(* CoDeSys 2.3.9.35 project: Exercício 8.pro *)
(* Author: Altus *)
(* Libraries: DU35x.lib 7.7.11 15:59:13, Navigation.lib 15.7.11 10:06:00, SysLibTargetVisu.lib 26.11.08 09:53:28, Standard.lib 26.11.08 09:46:20, Iecsfc.lib 26.11.08 09:46:14, SYSLIBCALLBACK.LIB 26.11.08 09:53:30 *)

(* PLC configuration (modules and I/O channels)
Configuração do CP [Root] node -1, in %IB0 out %QB0
  Comunicação [Comunica] node 0, in %IB0 out %QB0
    COM1 [COM1] node 0, in %IB0 out %QB0 {BaudRate = 115200; Paridade = Sem Paridade; StopBits = 1 Stop Bit; Modem = Sem RTS/CTS; Delay = 5}
      MToolIEC [Codesys] node 0, in %IB0 out %QB0
    COM2 [COM2] node 1, in %IB0 out %QB0 {BaudRate = 115200; Paridade = Sem Paridade; StopBits = 1 Stop Bit; Modem = Sem RTS/CTS; Delay = 5}
      Desabilitada [Desabilitado485] node 0, in %IB0 out %QB0
  Barramento [Barramento] node 1, in %IB0 out %QB0
    Entradas [Entradas] node 0, in %IB0 out %QB0
      Entradas Digitais 0 [Entradas0] node 0, in %IW0 out %QB0
        I00 AT %IX0.0 [BitInput] I0.0
        I01 AT %IX0.1 [BitInput] I0.1
        I02 AT %IX0.2 [BitInput] I0.2
        I03 AT %IX0.3 [BitInput] I0.3
        I04 AT %IX0.4 [BitInput] I0.4
        I05 AT %IX0.5 [BitInput] I0.5
        I06 AT %IX0.6 [BitInput] I0.6
        I07 AT %IX0.7 [BitInput] I0.7
        I08 AT %IX0.8 [BitInput] I0.8
      Entradas Digitais 1 [Entradas1] node 0, in %IW1 out %QB0
        I10 AT %IX1.0 [BitInput] I1.0
        I11 AT %IX1.1 [BitInput] I1.1
        I12 AT %IX1.2 [BitInput] I1.2
        I13 AT %IX1.3 [BitInput] I1.3
        I14 AT %IX1.4 [BitInput] I1.4
        I15 AT %IX1.5 [BitInput] I1.5
        I16 AT %IX1.6 [BitInput] I1.6
        I17 AT %IX1.7 [BitInput] I1.7
        I18 AT %IX1.8 [BitInput] I1.8
      Entradas Digitais 2 [Entradas2] node 0, in %IW2 out %QB0
        I20 AT %IX2.0 [BitInput] I2.0
        I21 AT %IX2.1 [BitInput] I2.1
      Entradas Analógicas [EntradaAnalogica] node 0, in %IW4 out %QB0
        AI0 AT %IW4 [WordInput] AI0 {TipoAnalogica = Channel Disable; FiltroAnalogica = Filter 0 - AI=2ms  / AV=90ms; FundoEscala = 0}
        AI1 AT %IW5 [WordInput] AI1 {TipoAnalogica = Channel Disable; FiltroAnalogica = Filter 0 - AI=2ms  / AV=90ms; FundoEscala = 0}
        AI2 AT %IW6 [WordInput] AI2 {TipoAnalogica = Channel Disable; FiltroAnalogica = Filter 0 - AI=2ms  / AV=90ms; FundoEscala = 0}
        AI3 AT %IW7 [WordInput] AI3 {TipoAnalogica = Channel Disable; FiltroAnalogica = Filter 0 - AI=2ms  / AV=90ms; FundoEscala = 0}
      Entradas Rápidas [EntradasRapidas] node 1, in %IB16 out %QB0
        Bloco 0 [Bloco0] node 0, in %IB16 out %QB0
          Desabilitado [DesabilitadoBloco0] node 0, in %IB16 out %QB0
        Bloco 1 [Bloco1] node 1, in %IB16 out %QB0
          Desabilitado [DesabilitadoBloco1] node 0, in %IB16 out %QB0
        Entrada Configuravél Bloco 0 [EntradaConfiBloco0] node 2, in %IB16 out %QB0
          Contador 0 [EntradaConfContador0] node 0, in %IB16 out %QB0 {EntradaConfiguravelContador = Disable}
        Entrada Configuravél Bloco 1 [EntradaConfiBloco1] node 3, in %IB16 out %QB0
          Contador 2 [EntradaConfContador2] node 0, in %IB16 out %QB0 {EntradaConfiguravelContador = Disable}
    Saídas [Saidas] node 1, in %IB13 out %QB0
      Saídas Digitais 0 [Saidas0] node 0, in %IW0 out %QW0
        Q00 AT %QX0.0 [BitOutput] Q0.0
        Q01 AT %QX0.1 [BitOutput] Q0.1
        Q02 AT %QX0.2 [BitOutput] Q0.2
        Q03 AT %QX0.3 [BitOutput] Q0.3
        Q04 AT %QX0.4 [BitOutput] Q0.4
        Q05 AT %QX0.5 [BitOutput] Q0.5
        Q06 AT %QX0.6 [BitOutput] Q0.6
        Q07 AT %QX0.7 [BitOutput] Q0.7
      Saídas Digitais 1 [Saidas1] node 0, in %IW0 out %QW1
        Q10 AT %QX1.0 [BitOutput] Q1.0
        Q11 AT %QX1.1 [BitOutput] Q1.1
        Q12 AT %QX1.2 [BitOutput] Q1.2
        Q13 AT %QX1.3 [BitOutput] Q1.3
        Q14 AT %QX1.4 [BitOutput] Q1.4
        Q15 AT %QX1.5 [BitOutput] Q1.5
        Q16 AT %QX1.6 [BitOutput] Q1.6
        Q17 AT %QX1.7 [BitOutput] Q1.7
      Saídas Analógicas [SaidaAnalogica] node 0, in %IW0 out %QW3
        AO0 AT %QW3 [WordOutput] AO0 {TipoAnalogica = Channel Disable; FundoEscala = 0}
        AO1 AT %QW4 [WordOutput] AO1 {TipoAnalogica = Channel Disable; FundoEscala = 0}
      Saídas Rápidas [SaidasRapidas] node 1, in %IB0 out %QB10
        Saída Rápida 0 Desabilitada [DesabilitadoF0] node 0, in %IB0 out %QB10
        Saída Rápida 1 Desabilitada [DesabilitadoF1] node 1, in %IB0 out %QB10
      Saídas Comum de Contador [SaidasContador] node 2, in %IB0 out %QB10
        Saída do Bloco 0 Desabilitada [DesabilitadoSaidaBloco0] node 0, in %IB0 out %QB10
        Saída do Bloco 1 Desabilitada [DesabilitadoSaidaBloco1] node 1, in %IB0 out %QB10
  Eventos Externos [Eventos] node 2, in %IB13 out %QB6
    Evento Temporizado [TimerEvent] node 0, in %IB13 out %QB6 {Intervalo = 10}
*)

(* Task configuration *)
TASK PRINCIPAL (PRIORITY := 1, INTERVAL := T#1ms);
	PLC_PRG();
END_TASK
TASK NAVIGATION (PRIORITY := 1, INTERVAL := T#20ms);
	NAVEGA();
END_TASK
TASK VISUALIZATION (PRIORITY := 1, INTERVAL := T#500ms);
	MAINTARGETVISU_PAINT_CODE
END_TASK
TASK KEYBOARD_USAGE (PRIORITY := 1, INTERVAL := T#20ms);
	MAINTARGETVISU_INPUT_CODE
END_TASK

(* POU PLC_PRG, ST *)
(*Um fulão processa o couro através do seguinte procedimento: A partir de um botão de início (entrada digital):
a) Inicialmente, preenche-se o fulão com o produto de curtimento, através da válvula VPC.
b) O motor é acionado no sentido horário, através da saída MH por um tempo THC.
c) O motor é acionado no sentido anti-horário, através da saída MAH, por um tempo TAHC.
d) O fulão é esvaziado, através da válvula VD.
e) O fulão é preenchido com água, através da válvula VL.
f) O motor é acionado no sentido horário, através da saída MH por um tempo THL.
g) O motor é acionado no sentido anti-horário, através da saída MAH, por um tempo TAHL.
h) O fulão é esvaziado, através da válvula VD.
i) É sinalizado, através de uma lâmpada FP, o final do processo.
Após o ciclo completo, o sistema deve ficar pronto para ser acionado novamente. O nível alto do fulão é indicado pela chave de
nível NVC, e o nível baixo (vazio) é indicado pela chave NVV. Elabore um programa que realize este procedimento, com os 
seguintes tempos para simulação: THC =TAHC= 5s. THL=TAHL=8s
Cada fase do processo deve ser devidamente apresentada na tela da IHM através de uma variável de texto.*)


PROGRAM PLC_PRG
VAR
	START AT %IX0.0: BOOL;
	NVC AT %IX0.1: BOOL; (*válvula que indica o nível alto do fulão*)
	NVV AT %IX0.2: BOOL; (*válvula que indica o nível baixo do fulão*)
	VPC AT %QX1.0: BOOL; (*válvula que inicia o preenchimento do fulão com produto de curtimento*)
	MH AT %QX1.1: BOOL; (*gira o motor no sentido horário*)
	MAH AT %QX1.2: BOOL; (*gira o motor no sentido anti-horário*)
	VD AT %QX1.3: BOOL; (*válvula que esvazia o fulão*)
	VL AT %QX1.4: BOOL; (*válvula que preenche o fulão com água*)
	FP AT %QX1.5: BOOL := 1; (*lâmpada que sinaliza quando o processo termina, começa acesa*)
	THC: TIME := T#5s; (*tempo que o motor fica girando no sentido horário, quando está esvaziando o fulão*)
	TAHC: TIME := T#5s; (*tempo que o motor fica girando no sentido anti-horário, quando está esvaziando o fulão*)
	THL: TIME := T#8s; (*tempo que o motor fica girando no sentido horário, quando está enchendo o fulão*)
	TAHL: TIME := T#8s; (*tempo que o motor fica girando no sentido anti-horário, quando está enchendo o fulão*)
	TH: TIME;
	TAH: TIME;
	T1: TON;
	T2: TON;
	B0: R_TRIG; (*borda de subida do botão de START*)
	B1: R_TRIG; (*borda de subida de NVC, que significa que chegou no nível alto do fulão*)
	B2: R_TRIG; (*borda de subida de NVV, que significa que chegou no nível baixo do fulão*)
	M1: INT := 0; (*variável de controle para o programa*)
	MSG: STRING(50) := 'DESLIGADO';
END_VAR
T1(IN := MH, PT := TH);
T2(IN := MAH, PT := TAH);
B0(CLK := START); (*borda de subida do botão de START*)
B1(CLK := NVC); (*borda de subida de NVC, que significa que chegou no nível ALTO do fulão*)
B2(CLK := NVV); (*borda de subida de NVV, que significa que chegou no nível BAIXO do fulão*)

IF B0.Q AND FP THEN (*quando der a borda de subida do botão de START*)
	FP := 0; (*desliga a lâmpada de FP, pois o processo se inicializou*)
	M1 := 1; (*iguala M1 a 1, que será usado depois*)
	VPC := 1; (*começa a enxer a válvula VPC, preenchendo o fulão com o produto de curtimento*)
	MSG := 'ENCHENDO O FULÃO COM PRODUTO DE CURTIMENTO';
END_IF

IF NOT FP THEN (*se a lâmpada estiver desligada, ou seja, não terminou o processo*)
	IF B1.Q THEN (*se chegou no nível alto do fulão*)
		IF VL THEN (*preencheu o fulão com água através da válvula VL*)
			VL := 0; (*desliga a válvula de água*)
			TH := THL; (*iguala o tempo de TH ao de THL, que é de 8 segundos*)
			TAH := TAHL; (*iguala o tempo de TAH ao de TAHL, que é de 8 segundos*)
		ELSE (*se encheu de produto de curtimento*)
			VPC := 0; (*desliga a válvula VPC de produto de curtimento, que para de mandar líquido para o fulão*)
			TH := THC; (*iguala o tempo de TH ao de THC, que é de 5 segundos*)
			TAH := TAHC; (*iguala o tempo de TAH ao de TAHC, que é de 5 segundos*)
		END_IF
		MH := 1; (*gira o motor no sentido horário por x segundos*)
		MSG := 'MOTOR GIRANDO NO SENTIDO HORÁRIO';
	END_IF
	IF T1.Q THEN (*quando acabar de contar o tempo de TH e der verdadeiro na saída T1.Q*)
		MH := 0; (*desliga a saída de MH*)
		MAH := 1; (*e aciona o motor no sentido anti-horário com a saída MAH por x segundos*)
		MSG := 'MOTOR GIRANDO NO SENTIDO ANTI-HORÁRIO';
	END_IF
	IF T2.Q THEN (*quando acabar de contar o tempo de TAHL e der verdadeiro na saída T2.Q*)
		MAH := 0; (*desliga a saída de MAH*)
		VD := 1; (*esvazia o fulão através da válvula VD*)
		MSG := 'ESVAZIANDO O FULÃO';
	END_IF
	IF B2.Q THEN (*se chegou no nível baixo do fulão*)
		VD := 0; (*desliga a válvula VD, para parar de esvaziar o fulão*)
		IF M1 = 1 THEN (*quando o botão de START é acionado, M1 é igualado a 1, então entra aqui depois*)
			M1 := M1 + 1; (*faz M1 + 1 e salva na própria variável de M1*)
			VL := 1; (*aciona a válvula de VL, para preencher o fulão com água*)
			MSG := 'PREENCHENDO O FULÃO COM ÁGUA';
		ELSE
			M1 := 0; (*iguala M1 a zero*)
			FP := 1; (*liga a lâmpada que indica que o fulão está cheio*)
			MSG := 'ACABOU O PROCESSO';
		END_IF
	END_IF
END_IF
END_PROGRAM

(* POU NAVEGA, ST *)
PROGRAM NAVEGA
VAR
	ControleTelas : NAVIGATION;
	ListaTelas 	: ARRAY [0..30] OF STRING(10);
END_VAR
(* Adiciona a tela MAIN como tela principal *)
ListaTelas[0] := 'MAIN';

(* Ativa o controle automático de navegação somente pelo teclado *)
ControleTelas(ENABLE_UPDW := FALSE, VISU_LIST := ListaTelas, UP := FALSE , DOWN := FALSE);
END_PROGRAM

(* Visualisation MAIN
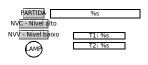
button at (9,6)-(30,16): text "PARTIDA"; toggles PLC_PRG.START
button at (5,17)-(34,26): text "NVC - Nível alto"; toggles PLC_PRG.NVC
button at (5,28)-(34,37): text "NVV - Nível baixo"; toggles PLC_PRG.NVV
ellipse at (11,39)-(28,55): text "LAMP"; alarm colour if PLC_PRG.FP
rectangle at (36,7)-(126,16): text "%s"; shows PLC_PRG.MSG
rectangle at (59,30)-(111,37): text "T1: %s"; shows PLC_PRG.T1.ET
rectangle at (59,40)-(111,47): text "T2: %s"; shows PLC_PRG.T2.ET
*)
